PROGRAM Device_rtrig
VAR
END_VAR

IO_Logs.bStartup_State(CLK := IO.bStartup_State );

IO_Logs.bStart(CLK := IO_control.bStart );
IO_Logs.bStop(CLK := IO_control.bStop );
IO_Logs.bReset(CLK := IO_control.bReset );
IO_Logs.bEstop(CLK := IO_control.bEstop );
IO_Logs.bOperational_State(CLK := IO.bOperational_State );

IO_Logs.data_send_flag(CLK := IO.data_send_flag );

IO_Logs.bConv1_In(CLK := IO.bConv1_In );
IO_Logs.bConv1_Out(CLK := IO.bConv1_Out);
IO_Logs.bConv2_In(CLK := IO.bConv2_In );
IO_Logs.bConv2_Out(CLK := IO.bConv2_Out);
IO_Logs.bConv3_In(CLK := IO.bConv3_In );
IO_Logs.bConv3_Out(CLK := IO.bConv3_Out);
IO_Logs.bConv4_In(CLK := IO.bConv4_In );
IO_Logs.bConv4_Out(CLK := IO.bConv4_Out);

END_PROGRAM

(* stored: Version 1.1.0.1, ProductVersion 3.1.4024.12
   POU Device_rtrig: Id {092b3d98-4634-4861-9cab-8539f287ebf9}, SpecialFunc None *)
